FUNCTION F_IsError : BOOL;
VAR_INPUT
	Feedback : I_CommandFeedback;
END_VAR

IF Feedback <> 0 AND_THEN Feedback.Error THEN
	F_IsError := TRUE;
END_IF

END_FUNCTION

(* stored: Version 1.1.0.1, ProductVersion 3.1.4024.12
   POU F_IsError: Id {7ddcec65-bcc6-0f23-0a72-12048093849f}, SpecialFunc None *)
